// TIA Portal V20 export
TYPE "UDT_Msg"
   STRUCT
      ID : Int;
      Number : DInt;
      Active : Bool;
      Level : Int;
   END_STRUCT;
END_TYPE
